FUNCTION_BLOCK InfluentSensors (* CAT Function Block Type *)
  (* Standard: 61499-2 *)
  (* Version 0.1, 10/7/2026, Claude/Hidryco, Schneider Electric, Rev1 - FeedReactorFlowPv (40FT05): QualityFailDelay = T#10s (tolerancia da falha de canal por qualidade do sinal Modbus) *)
  PACKAGE SE.Nereda;
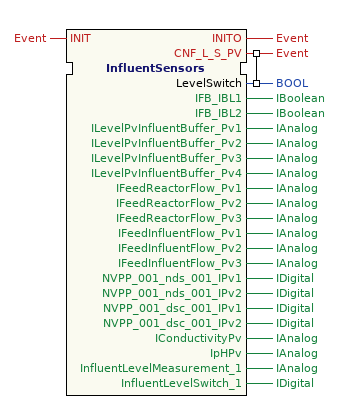
  EVENT_INPUT
    INIT; (* Initializes the symbolic link data destination FB with N (1 <= N <= 16) variables *)
  END_EVENT
  EVENT_OUTPUT
    INITO; (* Initialization Confirm *)
    CNF_L_S_PV WITH LevelSwitch; (* Execution confirmation of Pv *)
  END_EVENT
  VAR_OUTPUT
    LevelSwitch : BOOL; (* Process value output *)
  END_VAR
  PLUGS
    IFB_IBL1 : IBoolean;
    IFB_IBL2 : IBoolean;
  END_PLUGS
  PLUGS
    ILevelPvInfluentBuffer_Pv1 : IAnalog; (* Process value and status interface adapter *)
    ILevelPvInfluentBuffer_Pv2 : IAnalog; (* Process value and status interface adapter *)
    ILevelPvInfluentBuffer_Pv3 : IAnalog; (* Process value and status interface adapter *)
    ILevelPvInfluentBuffer_Pv4 : IAnalog; (* Process value and status interface adapter *)
    IFeedReactorFlow_Pv1 : IAnalog; (* Process value and status interface adapter *)
    IFeedReactorFlow_Pv2 : IAnalog; (* Process value and status interface adapter *)
    IFeedReactorFlow_Pv3 : IAnalog; (* Process value and status interface adapter *)
    IFeedInfluentFlow_Pv1 : IAnalog; (* Process value and status interface adapter *)
    IFeedInfluentFlow_Pv2 : IAnalog; (* Process value and status interface adapter *)
    IFeedInfluentFlow_Pv3 : IAnalog; (* Process value and status interface adapter *)
    NVPP_001_nds_001_IPv1 : IDigital; (* Process value interface adapter *)
    NVPP_001_nds_001_IPv2 : IDigital; (* Process value interface adapter *)
    NVPP_001_dsc_001_IPv1 : IDigital; (* Process value interface adapter *)
    NVPP_001_dsc_001_IPv2 : IDigital; (* Process value interface adapter *)
    IConductivityPv : IAnalog; (* Process value and status interface adapter *)
    IpHPv : IAnalog; (* Process value and status interface adapter *)
    InfluentLevelMeasurement_1 : IAnalog;
    InfluentLevelSwitch_1 : IDigital;
  END_PLUGS
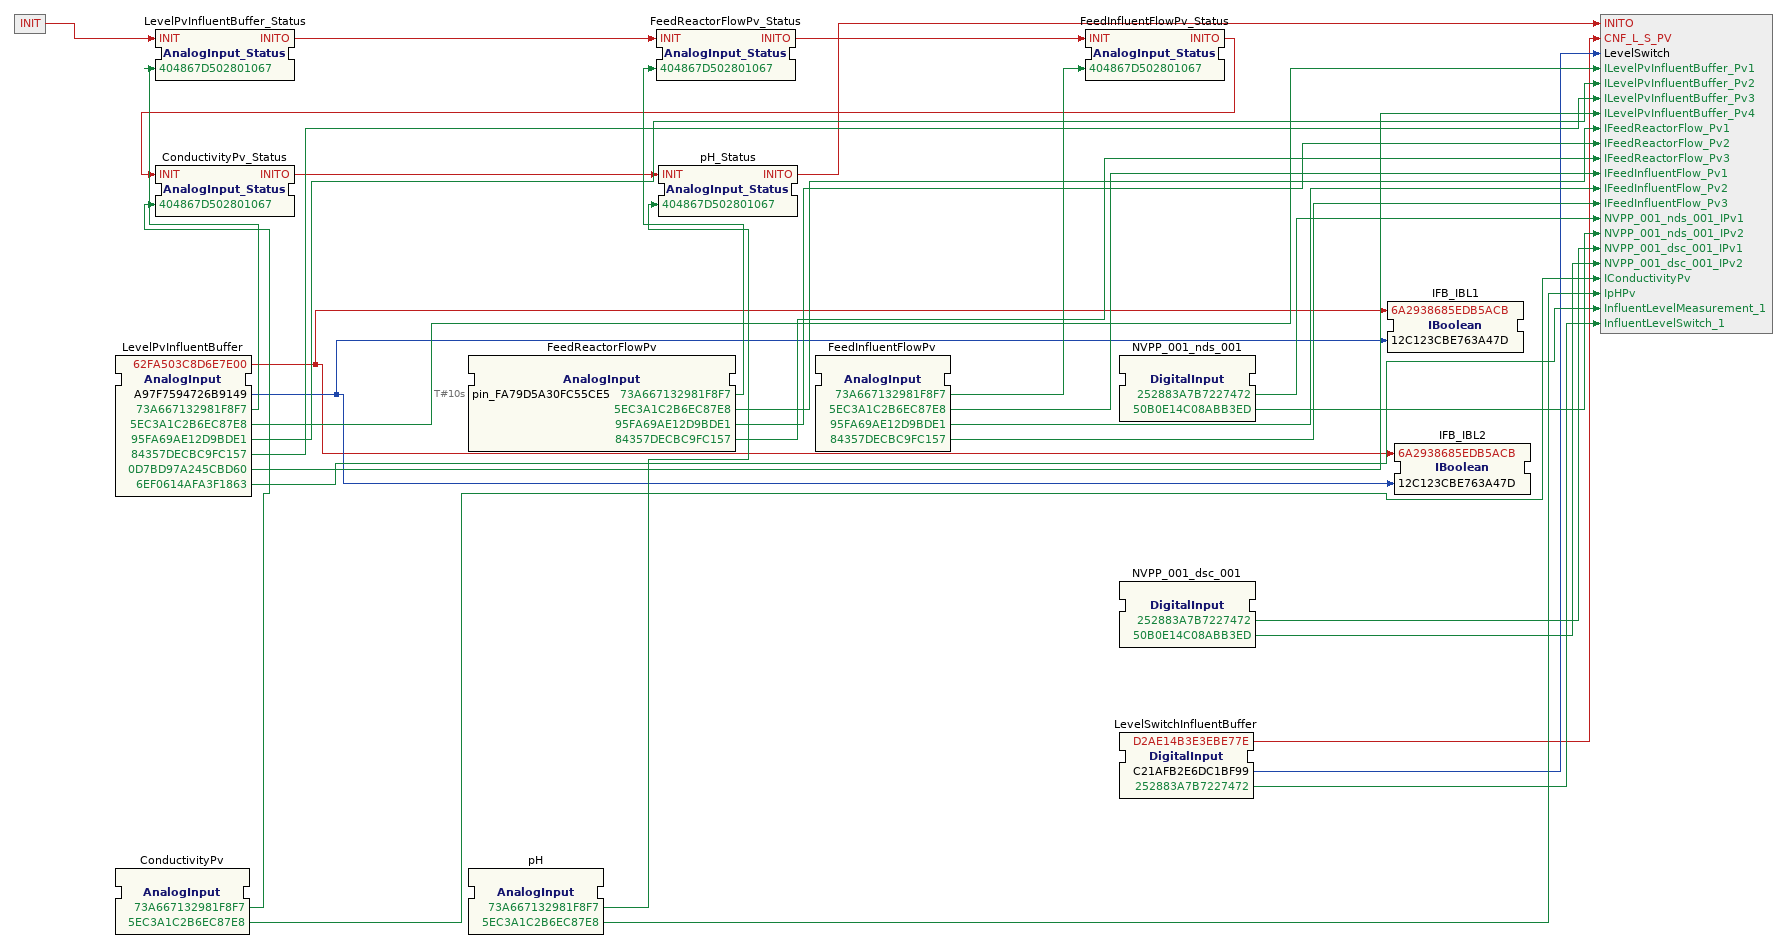
  (* 01 - FUNCTIONNAL INPUT INTERFACE *)
  (* 00 - INITIALIZATION *)
  (* 05 - LOGIC *)
  (* 06 - HMI INTERFACE *)
  (* 02 - FUNCTIONNAL OUTPUT INTERFACE *)
  (* Actuators Status *)
  (* 03 - FIELD INTERFACE *)
  (* Level measurement influent buffer *)
  (* Flow measurement reactor feed *)
  (* Flow measurement feed *)
  (* Conductivity measurement influent buffer *)
  (* pH measurement influent buffer *)
  FBS
    LevelPvInfluentBuffer_Status : AnalogInput_Status;
    FeedReactorFlowPv_Status : AnalogInput_Status;
    FeedInfluentFlowPv_Status : AnalogInput_Status;
    LevelPvInfluentBuffer : AnalogInput;
    FeedReactorFlowPv : AnalogInput(pin_FA79D5A30FC55CE5 := T#10s);
    FeedInfluentFlowPv : AnalogInput;
    NVPP_001_nds_001 : DigitalInput;
    NVPP_001_dsc_001 : DigitalInput;
    ConductivityPv : AnalogInput;
    pH : AnalogInput;
    ConductivityPv_Status : AnalogInput_Status;
    pH_Status : AnalogInput_Status;
    LevelSwitchInfluentBuffer : DigitalInput;
  END_FBS
  EVENT_CONNECTIONS
    LevelPvInfluentBuffer_Status.INITO TO FeedReactorFlowPv_Status.INIT;
    FeedReactorFlowPv_Status.INITO TO FeedInfluentFlowPv_Status.INIT;
    INIT TO LevelPvInfluentBuffer_Status.INIT;
    pH_Status.INITO TO INITO;
    ConductivityPv_Status.INITO TO pH_Status.INIT;
    FeedInfluentFlowPv_Status.INITO TO ConductivityPv_Status.INIT;
    LevelSwitchInfluentBuffer.D2AE14B3E3EBE77E TO CNF_L_S_PV;
    LevelPvInfluentBuffer.62FA503C8D6E7E00 TO IFB_IBL1.6A2938685EDB5ACB;
    LevelPvInfluentBuffer.62FA503C8D6E7E00 TO IFB_IBL2.6A2938685EDB5ACB;
  END_CONNECTIONS
  DATA_CONNECTIONS
    LevelSwitchInfluentBuffer.C21AFB2E6DC1BF99 TO LevelSwitch;
    LevelPvInfluentBuffer.A97F7594726B9149 TO IFB_IBL1.12C123CBE763A47D;
    LevelPvInfluentBuffer.A97F7594726B9149 TO IFB_IBL2.12C123CBE763A47D;
  END_CONNECTIONS
  ADAPTER_CONNECTIONS
    LevelPvInfluentBuffer.73A667132981F8F7 TO LevelPvInfluentBuffer_Status.404867D502801067;
    FeedReactorFlowPv.73A667132981F8F7 TO FeedReactorFlowPv_Status.404867D502801067;
    FeedInfluentFlowPv.73A667132981F8F7 TO FeedInfluentFlowPv_Status.404867D502801067;
    LevelPvInfluentBuffer.5EC3A1C2B6EC87E8 TO ILevelPvInfluentBuffer_Pv1;
    LevelPvInfluentBuffer.95FA69AE12D9BDE1 TO ILevelPvInfluentBuffer_Pv2;
    LevelPvInfluentBuffer.84357DECBC9FC157 TO ILevelPvInfluentBuffer_Pv3;
    FeedReactorFlowPv.5EC3A1C2B6EC87E8 TO IFeedReactorFlow_Pv1;
    FeedReactorFlowPv.95FA69AE12D9BDE1 TO IFeedReactorFlow_Pv2;
    FeedReactorFlowPv.84357DECBC9FC157 TO IFeedReactorFlow_Pv3;
    FeedInfluentFlowPv.5EC3A1C2B6EC87E8 TO IFeedInfluentFlow_Pv1;
    FeedInfluentFlowPv.95FA69AE12D9BDE1 TO IFeedInfluentFlow_Pv2;
    FeedInfluentFlowPv.84357DECBC9FC157 TO IFeedInfluentFlow_Pv3;
    NVPP_001_nds_001.252883A7B7227472 TO NVPP_001_nds_001_IPv1;
    NVPP_001_nds_001.50B0E14C08ABB3ED TO NVPP_001_nds_001_IPv2;
    NVPP_001_dsc_001.252883A7B7227472 TO NVPP_001_dsc_001_IPv1;
    NVPP_001_dsc_001.50B0E14C08ABB3ED TO NVPP_001_dsc_001_IPv2;
    LevelPvInfluentBuffer.0D7BD97A245CBD60 TO ILevelPvInfluentBuffer_Pv4;
    ConductivityPv.73A667132981F8F7 TO ConductivityPv_Status.404867D502801067;
    pH.73A667132981F8F7 TO pH_Status.404867D502801067;
    ConductivityPv.5EC3A1C2B6EC87E8 TO IConductivityPv;
    pH.5EC3A1C2B6EC87E8 TO IpHPv;
    LevelSwitchInfluentBuffer.252883A7B7227472 TO InfluentLevelSwitch_1;
    LevelPvInfluentBuffer.6EF0614AFA3F1863 TO InfluentLevelMeasurement_1;
  END_CONNECTIONS
END_FUNCTION_BLOCK
